TYPE ST_ValveDeadBand :
STRUCT
	fPosMax : LREAL := 29490.0;
	fPosMin : LREAL := 20950.0;
	fNegMax : LREAL := 18250.0;
	fNegMin : LREAL := 9830.0;
END_STRUCT
END_TYPE

(* stored: Version 1.1.0.1, ProductVersion 3.1.4024.12
   DUT ST_ValveDeadBand: Id {65c1e06a-9e6d-4b5b-b190-a7c17d54b243} *)
